{attribute 'GeneratedUsingTerminal: AT2041-0250-0020'}
{attribute addProperty BoxType "AT2041-0250-0020"}
{attribute addProperty Id "A_0102_AT2041_5250_0019_AT2041_5250AT2041_33A3DF1B80"}
{attribute addProperty CRC "1583719710"}
{attribute addProperty Size "80"}
{attribute addProperty Name "A_0042(AT2041-0250-0020)"}
TYPE A_0042_AT2041_0250_0020_5E65A51E EXTENDS AT2041_2EA6C9BF :
STRUCT
	{attribute addProperty Name "A_0102(AT2041-5250-0019) (AT2041-5250)"}
	{attribute addProperty PreviousPort "A_0042(AT2041-0250-0020) : B"}
	A_0102_AT2041_5250_0019_AT2041_5250 : AT2041_33A3DF1B;
END_STRUCT
END_TYPE

(* stored: Version 1.2.0.0, ProductVersion 3.1.4024.11
   DUT A_0042_AT2041_0250_0020_5E65A51E: Id {fa53f78c-9d8c-45ed-a57e-1a4977daa2cf} *)
